Xinje XDPPro project, PLC1: XL5E-16 (software 3.7.14b 2022-06-24)

PROGRAM 梯形图

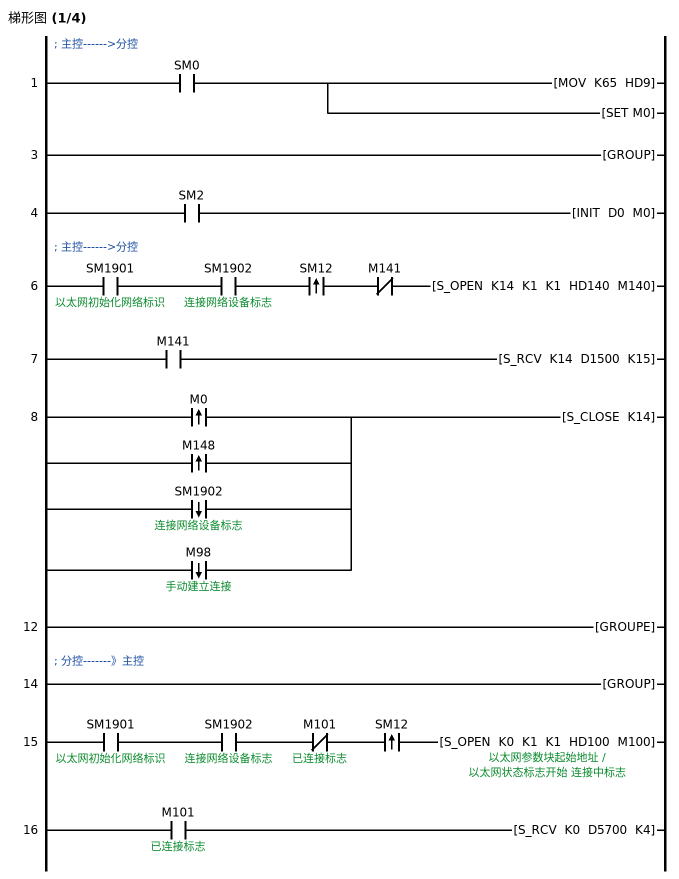
; 主控------>分控
LD     SM0
MOV    K65 HD9
SET    M0
GROUP
LD     SM2
INIT   D0 M0
; 主控------>分控
LD     SM1901	; 以太网初始化网络标识
AND    SM1902	; 连接网络设备标志
ANDP   SM12
ANI    M141
S_OPEN K14 K1 K1 HD140 M140
LD     M141
S_RCV  K14 D1500 K15
LDP    M0
ORP    M148
ORF    SM1902	; 连接网络设备标志
ORF    M98	; 手动建立连接
S_CLOSE K14
GROUPE
; 分控-------》主控
GROUP
LD     SM1901	; 以太网初始化网络标识
AND    SM1902	; 连接网络设备标志
ANI    M101	; 已连接标志
ANDP   SM12
S_OPEN K0 K1 K1 HD100 M100	; 以太网参数块起始地址 / 以太网状态标志开始 连接中标志
LD     M101	; 已连接标志
S_RCV  K0 D5700 K4

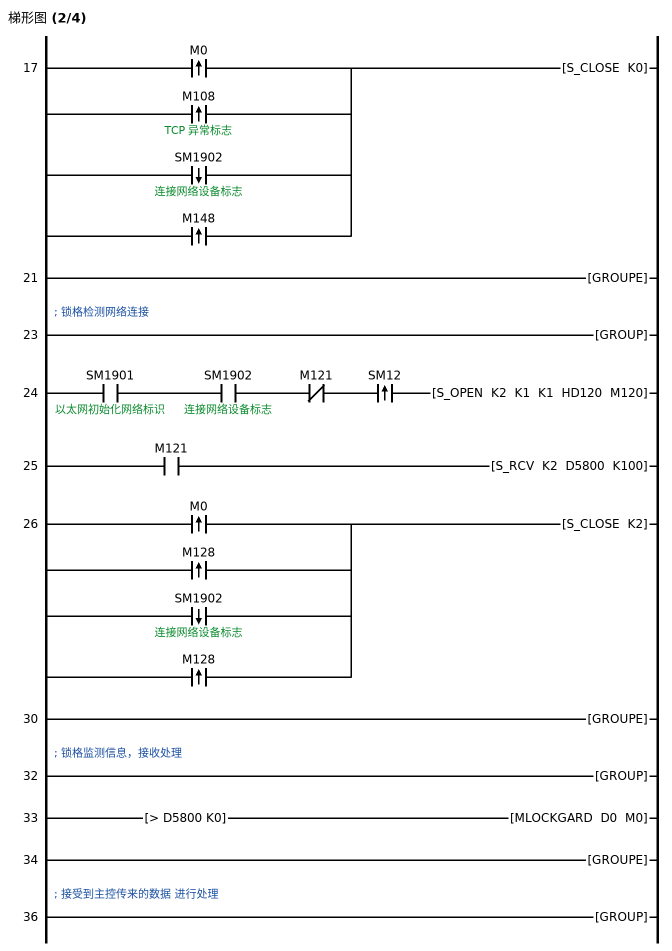
LDP    M0
ORP    M108	; TCP 异常标志
ORF    SM1902	; 连接网络设备标志
ORP    M148
S_CLOSE K0
GROUPE
; 锁格检测网络连接
GROUP
LD     SM1901	; 以太网初始化网络标识
AND    SM1902	; 连接网络设备标志
ANI    M121
ANDP   SM12
S_OPEN K2 K1 K1 HD120 M120
LD     M121
S_RCV  K2 D5800 K100
LDP    M0
ORP    M128
ORF    SM1902	; 连接网络设备标志
ORP    M128
S_CLOSE K2
GROUPE
; 锁格监测信息，接收处理
GROUP
LD>    D5800 K0
MLOCKGARD D0 M0
GROUPE
; 接受到主控传来的数据 进行处理
GROUP

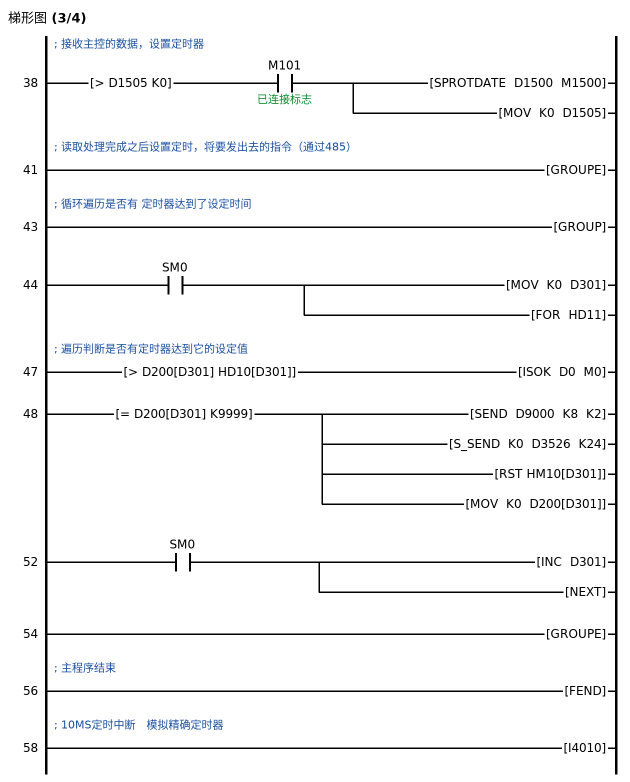
; 接收主控的数据，设置定时器
LD>    D1505 K0
AND    M101	; 已连接标志
SPROTDATE D1500 M1500
MOV    K0 D1505
; 读取处理完成之后设置定时，将要发出去的指令（通过485）
GROUPE
; 循环遍历是否有 定时器达到了设定时间
GROUP
LD     SM0
MOV    K0 D301
FOR    HD11
; 遍历判断是否有定时器达到它的设定值
LD>    D200[D301] HD10[D301]
ISOK   D0 M0
LD=    D200[D301] K9999
SEND   D9000 K8 K2
S_SEND K0 D3526 K24
RST    HM10[D301]
MOV    K0 D200[D301]
LD     SM0
INC    D301
NEXT
GROUPE
; 主程序结束
FEND
; 10MS定时中断　模拟精确定时器
I4010

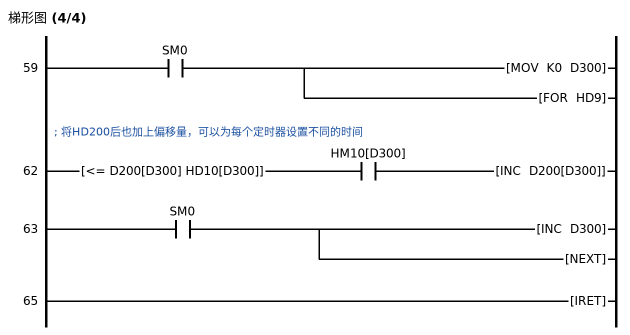
LD     SM0
MOV    K0 D300
FOR    HD9
; 将HD200后也加上偏移量，可以为每个定时器设置不同的时间
LD<=   D200[D300] HD10[D300]
AND    HM10[D300]
INC    D200[D300]
LD     SM0
INC    D300
NEXT
IRET

COMMENTS (devices not used above)
M95	上电关闭套接字
M109	错误标志
D202	485发送数据区
D201	485发送数据长度
D999	发送区首地址偏移量
T0	等待100ms再开启接受
M99	已开启以太网接受标志
D220	485发送数据区结束
D100	以太网接受数据存储开始
D119	以太网接受数据存储区结束
M96	以太网接受数据
M97	以太网发送数据
M102	发送中标志
M103	已发送标志
M104	接收中标志
M105	已接收标志
M106	关闭中标志
M107	MODBUS TCP 通信中标志
M2000	小车控制定时器
M1999	处理完成标志
D2000	模拟定时器发送缓冲区首地址
D1601	数据开始区
D3000	小车入格定时器定时值
M3000	小车入格定时器 开启标志
D1000	发送缓冲区地址的临时变量
M110	0号套接字已连接标注
D303	485接收缓冲区步进值
D5000	485接收缓冲区
M1511	小车落格成功后回传数据给主控
D9700	记录当前分支触发次数用

C FUNCTION BLOCK return485.fcb
/* 当电滚筒返回数据时进行处理
1.电滚筒运行成功，则向主控返回成功信息
2.电滚筒运行失败，向主控返回电滚筒错误信息
#EXPORT_ENTRY_BEGIN(RETURN485)
//    类型              模式             个数               映射          注释
W = { type = "PINT16S", mode = [In,Out], count = "unknown", map = [D,HD], comment = "" }
B = { type = "BIT"    , mode = [In,Out], count = "unknown", map = [M,HM], comment = "" }
#EXPORT_ENTRY_END */
/*************************************************************************
 * FunctionBlockName:  RETURN485
 * Version:            1.0.0
 * Author:             rpl
 * UpdateTime:         2022-09-04 14:31:17
 * Comment:            当电滚筒返回数据时进行处理
1.电滚筒运行成功，则向主控返回成功信息
2.电滚筒运行失败，向主控返回电滚筒错误信息
**************************************************************************/

/**
 * @summary 
 * @param W 
 * @param B 
 */
 //D5000为接收区首地址
void RETURN485(PINT16S W,BIT B)
{
    #define SysRegAddr_HD_D_HM_M
    /***通过按位与操作得出不同的情况***/
    /*分别处理四个字节的数据*/
    
    //第二个,通过左移动右移动得到小车号
    D[5001] = D[5001] << 11;
    D[5001] = D[5001] >> 11;
    
    //第三位
    if ( D[5002] )
    {
        //大于零表示存在故障,直接将故障码上报，现场操作人员根据故障码得到具体错误信息
        //数据存入小车对应状态数组后直接返回，不做后续处理
        D[10000+D[5001]] = D[5002] ;
        return;
    }
    //第四位校验位暂不处理
    
    
    /*********************处理将要回传给主控plc的信息***************************/
    /**从D3526开始*/
    D[3526] = 0x02;
    D[3527] = 5;
    
    /**报文编号 8个寄存器 acsii码形式**/
    D[3528] = 48;
    D[3529] = 49;
    D[3530] = 50;
    D[3531] = 51;
    D[3532] = 52;
    D[3533] = 53;
    D[3534] = 54;
    D[3535] = 55;
    
    /******小车编号 四个寄存器 千百十个， 千位和百位直接设为0*******/
    
    D[3536] = 48;
    D[3537] = 48;
    D[3538] = ( D[5001] / 10 ) % 10;
    D[3539] = D[5001] % 10;
    
    /******实际落袋格口 4个字节**********/
    D[3540] = 48;
    D[3541] = 48;
    D[3542] = ( D[50050 + D[5001]] / 10 ) % 10;
    D[3543] = D[50050 + D[5001]] % 10;
    
    /********补5个空格***********/
    D[3544] = 32;
    D[3545] = 32;
    D[3546] = 32;
    D[3547] = 32;
    D[3548] = 32;
    
    /*****结束符*****/
    D[3549] = 0x03;
    
    /*******发送触发************/
    M[1511] = 1;

    
}

C FILE func1.h
#ifndef	_FUNC1_H
#define	_FUNC1_H

/*******配置数据******************/
#define  GardNum  60   //格口数量
#define CarNum    60    //小车数量
#define CarLowLine     40   //小车号下限
#define CarHighLine    80   //小车号上限
#define ALLTIME  40000  //运行一圈的时间
/*****占用长度******/
#define TimerBufferSize 10

/***小车数据结构体**/
typedef struct{

INT16U Car_Mark;       //小车号
int  Destination[4]; //格口数组
INT16U NeedTime[4]; //时间数组
INT16U Master; //命令语
int NOW; //步进值
    
} Car_Date;


/***待投放小车数据**/ 
 Car_Date AwaitQueue[CarNum];


/***锁格数组***/
INT16S LockGard[GardNum];


/***定时器发送缓冲区***/



/***********各个结构体或数组的首地址***********/
#define LockGard_FirstAdress   D+5000
#define Car_Date_FirstAdress   D+5100
#define AwaitQueue_FirstAdress D+4500 
#define SendBuffer485           D+9000


#endif

C FUNCTION BLOCK isok.fcb
/* 检查将要落下的格口有没有锁格，如果有就找其他的可以下的格口，如果仅有这一个则再转一圈再下
#EXPORT_ENTRY_BEGIN(ISOK)
//    类型              模式             个数               映射          注释
W = { type = "PINT16S", mode = [In,Out], count = "unknown", map = [D,HD], comment = "" }
B = { type = "BIT"    , mode = [In,Out], count = "unknown", map = [M,HM], comment = "" }
#EXPORT_ENTRY_END */
/*************************************************************************
 * FunctionBlockName:  ISOK
 * Version:            1.0.0
 * Author:             rpl
 * UpdateTime:         2022-09-03 16:23:50
 * Comment:            检查将要落下的格口有没有锁格,如果有就找其他的可以下的格口,如果仅有这一个则再转一圈再下
**************************************************************************/

/**
 * @summary
 * @param W
 * @param B
 */

#include"func1.h"
#define SendFirstAddress 3526
// 锁格数组 D50000 -D50099  暂定为50个
//小车对应格口 D50100- D50199 暂定位100个
//D[301]是定时器及其发送缓冲区偏移量
void ISOK ( PINT16S W, BIT B )
{
#define SysRegAddr_HD_D_HM_M_SD


/************************************判断是否锁格**********************************/


   if( LockGard[D[2008 + D[301] * TimerBufferSize]] ==1)
    {
    //该格口被锁住了,寻找下一个适合的格口,将定时器的值重置D[200+D[301]] HD [200+D[301]]
    Car_Date* TempCarDate = Car_Date_FirstAdress + D[301] * sizeof ( Car_Date )/2 ;
    
    (TempCarDate->NOW)++;
    if(TempCarDate->NOW >3)
    {
        TempCarDate->NOW = 0;
    }
    D [200 + D[301]] = 0;
    HD[200 + D[301]] = TempCarDate->NeedTime[TempCarDate->NOW];
    //实际落格格口号
    D[2008 + D[301]*TimerBufferSize] = TempCarDate->Destination[TempCarDate->NOW];
    

    

    return;
    }


//}
    /***暂不确定在FOR循环中是否不支持类似D2000[D9998]类似的偏移操作还是另有原因
        在该函数中将数据转运到一个固定的发送缓冲区地点。
    ***/
    /************************************485发送指令**********************************/
    int tmp =  D[301] * TimerBufferSize;
    * ( SendBuffer485  ) = D[2000 + tmp];
    * ( SendBuffer485 + 1 ) = D[2001 + tmp];
    * ( SendBuffer485 + 2 ) = D[2002 + tmp];
    * ( SendBuffer485 + 3 ) = D[2003 + tmp];
    * ( SendBuffer485 + 4 ) = D[2004 + tmp];
    * ( SendBuffer485 + 5 ) = D[2005 + tmp];
    * ( SendBuffer485 + 6 ) = D[2006 + tmp];
    * ( SendBuffer485 + 7 ) = D[2007 + tmp];

    D[9998] = D[301] * TimerBufferSize;
    D[200 + D[301]] = 9999;
    M[1512] = 1;
    
    /******************************返回主控分拣完成*****************************************/
    
    
    //第一个寄存器，小车发送起始符号
	
	//第二个寄存器，应答的小车编号
    
	
	
	/****得到小车编号,落袋格口号****/
    INT16U mcarmark = D[2009 + tmp];
    INT16U mdestination = D[2008 +tmp]; //存在错误,无法准确知道小车在哪儿下了

        //除2的原因，1byte=8bit 一个寄存器=2个byte
        //Car_Date* TempCarDate = Car_Date_FirstAdress + i * sizeof ( Car_Date )/2 ;

     //起始符
     D[SendFirstAddress] = 0x02;
     //命令语
     D[SendFirstAddress + 1] = 53;
     //报文编号
     D[SendFirstAddress + 2] = 48 + SD[13]%10;
     D[SendFirstAddress + 3] = 48+(SD[13]/10)%10;
     D[SendFirstAddress + 4] = 48 + SD[14]%10;
     D[SendFirstAddress + 5] = 48 + (SD[14]/10)%10;
     D[SendFirstAddress + 6] = 48+SD[15]%10;
     D[SendFirstAddress + 7] = 48+(SD[15]/10)%10;
     D[SendFirstAddress + 8] = 48 + SD[16]%10;
     D[SendFirstAddress + 9] = 48 + mcarmark%10 ;
     //小车号
     D[SendFirstAddress + 10] = 48; //千位
     D[SendFirstAddress + 11] = 48+( mcarmark / 100 ) % 10;//百位
     D[SendFirstAddress + 12] = 48 + ( mcarmark / 10 ) % 10; //十位
     D[SendFirstAddress + 13] = 48 + ( mcarmark % 10 );//个位
     //实际落袋格口号
     D[SendFirstAddress + 14] = 48;
     D[SendFirstAddress + 15] = 48 + ( mdestination/ 100 ) % 10;
     D[SendFirstAddress + 16] = 48 + ( mdestination / 10 ) % 10;
     D[SendFirstAddress + 17] = 48 + ( mdestination ) % 10;
     //5位空格
     D[SendFirstAddress + 18] = 32;
     D[SendFirstAddress + 19] = 32;
     D[SendFirstAddress + 20] = 32;
     D[SendFirstAddress + 21] = 32;
     D[SendFirstAddress + 22] = 32;
     //结束符
     D[SendFirstAddress + 23] = 0x03;
 
    
    return;
}

C FUNCTION BLOCK mlockgard.fcb
/* #EXPORT_ENTRY_BEGIN(MLOCKGARD)
//    类型              模式             个数               映射          注释
W = { type = "PINT16S", mode = [In,Out], count = "unknown", map = [D,HD], comment = "" }
B = { type = "BIT"    , mode = [In,Out], count = "unknown", map = [M,HM], comment = "" }
#EXPORT_ENTRY_END */
/*************************************************************************
 * FunctionBlockName:  MLOCKGARD
 * Version:            1.0.0
 * Author:             
 * UpdateTime:         2022-09-13 16:42:11
 * Comment:            
**************************************************************************/

/**
 * @summary 
 * @param W 
 * @param B 
 */
 #include"func1.h"
void MLOCKGARD(PINT16S W,BIT B)
{
	#define SysRegAddr_HD_D_HM_M 
	
	for(int i =0;i<GardNum;i++)
	{
        LockGard[i] = D[5801 + i];
	}

return;
}

C FUNCTION BLOCK sprotdate.fcb
/* 处理上位机发来的具体控制信息，得到需要的指令
#EXPORT_ENTRY_BEGIN(SPROTDATE)
//    类型              模式             个数               映射          注释
W = { type = "PINT16S", mode = [In,Out], count = "unknown", map = [D,HD], comment = "" }
B = { type = "BIT"    , mode = [In,Out], count = "unknown", map = [M,HM], comment = "" }
#EXPORT_ENTRY_END */
/*************************************************************************
 * FunctionBlockName:  SPROTDATE
 * Version:            1.0.0
 * Author:             plc
 * UpdateTime:         2022-09-03 11:25:44
 * Comment:            处理上位机发来的具体控制信息，得到需要的指令
**************************************************************************/

/**
 * @summary 
 * @param W 
 * @param B 
 */
 
 #include"func1.h"
#define _Command       D[92]
#defien RCVFromMainAddress    D+1500
/******当前分控所控制的小车上下限**********/
#define CarLowLine     40
#define CarHighLine    80


void SPROTDATE(PINT16S W,BIT B)
{
	#define SysRegAddr_HD_D_HM_M
	/*******首先判断小车号是否是当前分控plc所管辖的*******/
	 INT16U _Car_Mark    = *(RCVFromMainAddress+13);      //小车号
	 if(_Car_Mark <= CarLowLine || _Car_Mark > CarHighLine) 
    {
     /***如果不是，直接退出程序***/
        return;
    }
	
	INT16U _Runtime1，_Runtime2，_Runtime3，_Runtime4；
	INT16U _Destination1，_Destination2，_Destination3，_Destination4；
	 /*******************拼接时间****************/
     *(RCVFromMainAddress+1)= *(RCVFromMainAddress+1) << 8; 
    _Runtime1  = *(RCVFromMainAddress+1) + *(RCVFromMainAddress+2);      //定时器时间毫秒为单位
    
    *(RCVFromMainAddress+3) = *(RCVFromMainAddress+3) << 8;
    _Runtime2 = *(RCVFromMainAddress+3) + *(RCVFromMainAddress+4);
    
    *(RCVFromMainAddress+5) = *(RCVFromMainAddress+5) << 8;
    _Runtime3 = *(RCVFromMainAddress+5) + *(RCVFromMainAddress+6);
    
    *(RCVFromMainAddress+7) = *(RCVFromMainAddress+7) << 8;
    _Runtime4 = *(RCVFromMainAddress+7) + *(RCVFromMainAddress+8);
    /*************写入格口号*********************/
    _Destination1 = *(RCVFromMainAddress+9);
    _Destination2 = *(RCVFromMainAddress+10);
    _Destination3 = *(RCVFromMainAddress+11);
    _Destination4 = *(RCVFromMainAddress+12);
    
    _Command     = *(RCVFromMainAddress+14);      //命令语
    //找到小车数组，将信息写入小车数组对应的对象中


        Car_Date* TempCarDate = Car_Date_FirstAdress + (_Car_Mark-41) * sizeof ( Car_Date )/2 ;
        if(TempCarDate->Car_Mark ==  _Car_Mark)
        {
            TempCarDate->Destination[0] =  _Destination1;
            TempCarDate->NeedTime[0] = _Runtime1;
            TempCarDate->Destination[1] =  _Destination2;
            TempCarDate->NeedTime[1] = _Runtime2;
            TempCarDate->Destination[2] =  _Destination3;
            TempCarDate->NeedTime[2] = _Runtime3;
            TempCarDate->Destination[3] =  _Destination4;
            TempCarDate->NeedTime[3] = _Runtime4;
            TempCarDate->Master   = _Command;
        }
    
/**************************************************根据指令进行处理**************************************************/
	switch(_Command)
	{
	  //分拣指令
	  
	 case 49: 
        //1.设置定时器
        //2.处理要发给的小车指令 485通讯
        

        /**指向该小车专用定时器**/
   
                
                //为该定时器发送缓冲区写入数据.每个缓冲区为8个寄存器
                D[2000 + _Car_Mark * TimerBufferSize] = 0x94;     //帧头
                //方向以及小车编号
                if ( _Destination1 % 2 )
                {
                    D[2001 + _Car_Mark * TimerBufferSize] = 32+_Car_Mark-40;
                
                }
                else
                {
                    D[2001 + _Car_Mark * TimerBufferSize] = 96 + _Car_Mark-40;
                }
                
                D[2002 + _Car_Mark * 10] = 0x7F;    //运行速度低七位
                D[2003 + _Car_Mark * TimerBufferSize] = 0x00;     //延迟运行时间第七位
                D[2004 + _Car_Mark * TimerBufferSize] = 0x7F;     //运行时间低七位
                D[2005 + _Car_Mark * TimerBufferSize] = 0x4E;     //复合数据：位置或时间控制模式，距离或时间第八位，延迟时间第八位
                D[2006 + _Car_Mark * TimerBufferSize] = 0x32;     //复合数据二
                D[2007 + _Car_Mark * TimerBufferSize] = ( (D[2001 + _Car_Mark * TimerBufferSize]) ^ (D[2002 + _Car_Mark * TimerBufferSize] )^ (D[2003 + _Car_Mark * TimerBufferSize]) ^ (D[2004 + _Car_Mark * TimerBufferSize]) ^ (D[2005 + _Car_Mark * TimerBufferSize]) ^ (D[2006 + _Car_Mark * TimerBufferSize]) ) & (0x7F); //校验位
                
                //存储格口号 和小车号 
                D[2008 + _Car_Mark * TimerBufferSize]   = _Destination1;
                D[2009 + _Car_Mark * TimerBufferSize]    =   _Car_Mark;
                /**设置完一个就退出循环**/	 
                HD[10 + _Car_Mark] = _Runtime1;   //设置定时时间
                HM[10 + _Car_Mark] = 1;        //开启定时器
        break;
        
        
      //齐格指令 
	 case 50:
        break;
        
     //锁格指令
	 case 51:
        break;
        
	}

}

C FUNCTION BLOCK init.fcb
/* #EXPORT_ENTRY_BEGIN(INIT)
//    类型              模式             个数               映射          注释
W = { type = "PINT16S", mode = [In,Out], count = "unknown", map = [D,HD], comment = "" }
B = { type = "BIT"    , mode = [In,Out], count = "unknown", map = [M,HM], comment = "" }
#EXPORT_ENTRY_END */
/*************************************************************************
 * FunctionBlockName:  INIT
 * Version:            1.0.0
 * Author:             RPL
 * UpdateTime:         2022-09-05 14:03:56
 * Comment:            
**************************************************************************/

/**
 * @summary 
 * @param W 
 * @param B 
 */
 #include"func1.h"
void INIT(PINT16S W,BIT B)
{
	#define SysRegAddr_HD_D_HM_M
	
	//初始化小车数组
	for(int i = 0; i<CarNum;i++)
    {
        
      (( Car_Date * ) ( Car_Date_FirstAdress + i * sizeof ( Car_Date )/2 ))->Car_Mark = i + 1;
    }
	//初始化锁格数组
	for(int i = 0 ; i <= GardNum; i++)
	{
        LockGard[i] = 0;
	}
	
	
	

}

C FUNCTION BLOCK control.fcb
/* #EXPORT_ENTRY_BEGIN(CONTROL)
//    类型              模式             个数               映射          注释
W = { type = "PINT16S", mode = [In,Out], count = "unknown", map = [D,HD], comment = "" }
B = { type = "BIT"    , mode = [In,Out], count = "unknown", map = [M,HM], comment = "" }
#EXPORT_ENTRY_END */
/*************************************************************************
 * FunctionBlockName:  CONTROL
 * Version:            1.0.0
 * Author:             RPL
 * UpdateTime:         2022-09-05 10:46:15
 * Comment:            
**************************************************************************/

/**
 * @summary 
 * @param W 
 * @param B 
 */
 #include"func1.h"
 
 #define RCV_FirstAddress D+5000
 /*接收到电滚筒返回的数据之后，处理一下然后返回给主控，主控直接返回给上位机
    需要返回24个字节的数据 起始位置为D3526
 
 */
 
 //接收起始地址为D5000 4个寄存器
void CONTROL(PINT16S W,BIT B)
{
	#define SysRegAddr_HD_D_HM_M
	


}